FUNCTION_BLOCK FB_TestMCSimple EXTENDS CL_HystoDebug
VAR
  stm	: UINT := 10;
  bMCRun, bFW, bBW,bPower,bReset,bResetDone,bError,bBusy,bPowerStatus : BOOL := FALSE;
  errId : UDINT;
  
  fbPower : MC_Power;
  fbReset : MC_Reset;
END_VAR

fbPower(
	Axis:= G.stAX.Line1Front, 
	Enable:= bPower, 
	Enable_Positive:= bPower, 
	Enable_Negative:= bPower, 
	Override:= 100.0, 
  Status=>bPowerStatus,
	Busy=>bBusy , 
	Error=>bError, 
	ErrorID=> errId);

fbReset(
	Axis:= G.stAX.Line1Front, 
	Execute:= bReset, 
	Done=> bResetDone,
	Busy=> bBusy, 
	Error=>bError, 
	ErrorID=>errId);
  
CASE stm OF 
  1:
		bPower := TRUE;
    bMCRun := TRUE;
		stm := 2;
	2:
		IF G.stAX.Line1Front.Status.Error THEN //really at the level of NC
			stm := 3;
		ELSE
			stm := 5;
		END_IF
	3:
		bReset := TRUE;
		stm := 4;	
	4:
		IF bResetDone THEN
			bReset := FALSE;
			stm := 5;
		END_IF
	5:
    bPowerStatus := fbPower.Status;
		IF bPowerStatus THEN
			stm := 6;
		END_IF
  6:
    stm := 6;
end_case

END_FUNCTION_BLOCK

(* stored: Version 1.1.0.1, ProductVersion 3.1.4024.12
   POU FB_TestMCSimple: Id {0630e2cf-2446-4a55-9ef4-978bf9a13065}, SpecialFunc None *)
